# EPICS substitutions: db/Beckhoff_MX/ecmcMB1120.substitutions
#- MB1120 is a passive backplane junction and exposes no process data.
file "empty.template" {
  pattern {}
}
